// TIA Portal V20 export
FUNCTION "02 T4 LANT HMI" : Void   // FC1212, LAD
TITLE = HMI
{ S7_Optimized_Access := 'TRUE' }
// stored: AutoNumber false, SetENOAutomatically false
BEGIN

REGION Network 1: Reset command interface from HMI in case of time-out
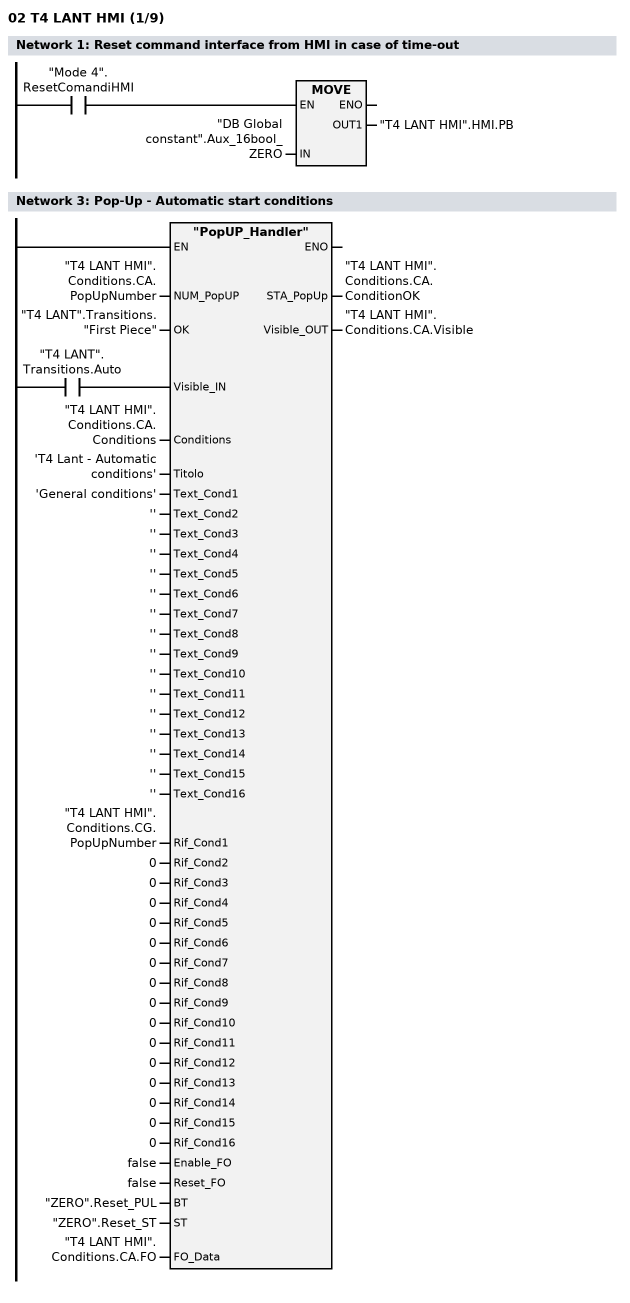
   RUNG wire#powerrail
      Contact( "Mode 4".ResetComandiHMI )
      Move(in := "DB Global constant".Aux_16bool_ZERO, out1 => "T4 LANT HMI".HMI.PB)
   END_RUNG
   // the same network as SCL:
   IF "Mode 4".ResetComandiHMI THEN "T4 LANT HMI".HMI.PB := "DB Global constant".Aux_16bool_ZERO; END_IF;
END_REGION

REGION Network 2: ============ POP UP ============
END_REGION

REGION Network 3: Pop-Up - Automatic start conditions
   RUNG wire#powerrail
      "PopUP_Handler"(Visible_IN := wire#w1, NUM_PopUP := "T4 LANT HMI".Conditions.CA.PopUpNumber, OK := "T4 LANT".Transitions."First Piece", Conditions := "T4 LANT HMI".Conditions.CA.Conditions, Titolo := 'T4 Lant - Automatic conditions', Text_Cond1 := 'General conditions', Text_Cond2 := '', Text_Cond3 := '', Text_Cond4 := '', Text_Cond5 := '', Text_Cond6 := '', Text_Cond7 := '', Text_Cond8 := '', Text_Cond9 := '', Text_Cond10 := '', Text_Cond11 := '', Text_Cond12 := '', Text_Cond13 := '', Text_Cond14 := '', Text_Cond15 := '', Text_Cond16 := '', Rif_Cond1 := "T4 LANT HMI".Conditions.CG.PopUpNumber, Rif_Cond2 := 0, Rif_Cond3 := 0, Rif_Cond4 := 0, Rif_Cond5 := 0, Rif_Cond6 := 0, Rif_Cond7 := 0, Rif_Cond8 := 0, Rif_Cond9 := 0, Rif_Cond10 := 0, Rif_Cond11 := 0, Rif_Cond12 := 0, Rif_Cond13 := 0, Rif_Cond14 := 0, Rif_Cond15 := 0, Rif_Cond16 := 0, Enable_FO := false, Reset_FO := false, BT := "ZERO".Reset_PUL, ST := "ZERO".Reset_ST, FO_Data := "T4 LANT HMI".Conditions.CA.FO, STA_PopUp => "T4 LANT HMI".Conditions.CA.ConditionOK, Visible_OUT => "T4 LANT HMI".Conditions.CA.Visible)
   END_RUNG
   RUNG wire#powerrail
      Contact( "T4 LANT".Transitions.Auto )
   END_RUNG wire#w1
   // the same network as SCL:
   "PopUP_Handler"(NUM_PopUP := "T4 LANT HMI".Conditions.CA.PopUpNumber,
                   OK := "T4 LANT".Transitions."First Piece",
                   Visible_IN := "T4 LANT".Transitions.Auto,
                   Conditions := "T4 LANT HMI".Conditions.CA.Conditions,
                   Titolo := 'T4 Lant - Automatic conditions',
                   Text_Cond1 := 'General conditions',
                   Text_Cond2 := '',
                   Text_Cond3 := '',
                   Text_Cond4 := '',
                   Text_Cond5 := '',
                   Text_Cond6 := '',
                   Text_Cond7 := '',
                   Text_Cond8 := '',
                   Text_Cond9 := '',
                   Text_Cond10 := '',
                   Text_Cond11 := '',
                   Text_Cond12 := '',
                   Text_Cond13 := '',
                   Text_Cond14 := '',
                   Text_Cond15 := '',
                   Text_Cond16 := '',
                   Rif_Cond1 := "T4 LANT HMI".Conditions.CG.PopUpNumber,
                   Rif_Cond2 := 0,
                   Rif_Cond3 := 0,
                   Rif_Cond4 := 0,
                   Rif_Cond5 := 0,
                   Rif_Cond6 := 0,
                   Rif_Cond7 := 0,
                   Rif_Cond8 := 0,
                   Rif_Cond9 := 0,
                   Rif_Cond10 := 0,
                   Rif_Cond11 := 0,
                   Rif_Cond12 := 0,
                   Rif_Cond13 := 0,
                   Rif_Cond14 := 0,
                   Rif_Cond15 := 0,
                   Rif_Cond16 := 0,
                   Enable_FO := false,
                   Reset_FO := false,
                   BT := "ZERO".Reset_PUL,
                   ST := "ZERO".Reset_ST,
                   FO_Data := "T4 LANT HMI".Conditions.CA.FO,
                   STA_PopUp => "T4 LANT HMI".Conditions.CA.ConditionOK,
                   Visible_OUT => "T4 LANT HMI".Conditions.CA.Visible);
END_REGION

REGION Network 4: Pop- Up - General conditions
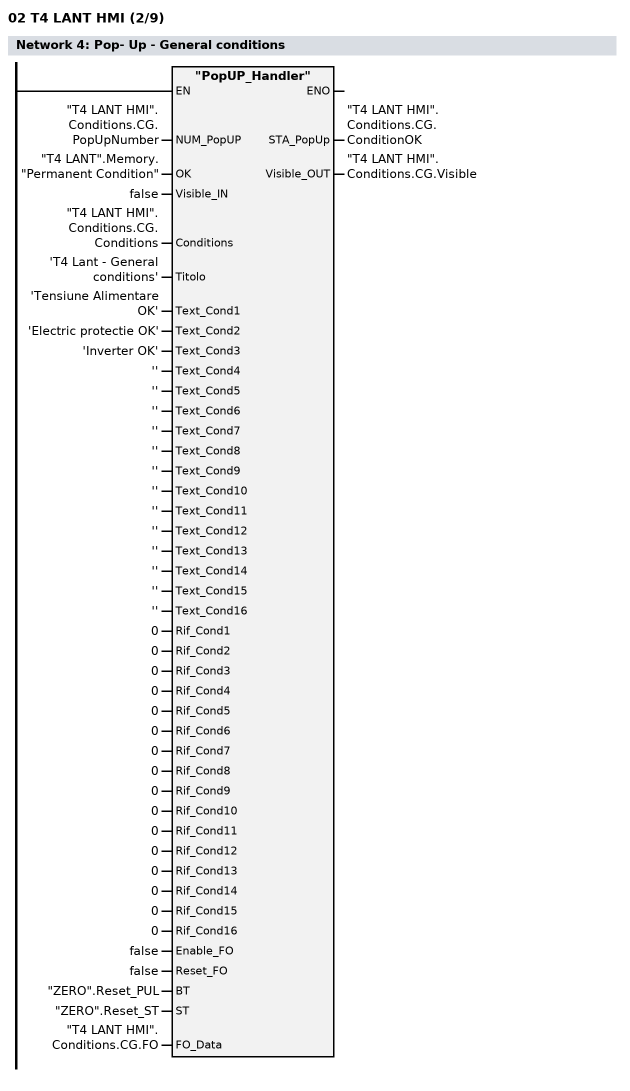
   RUNG wire#powerrail
      "PopUP_Handler"(NUM_PopUP := "T4 LANT HMI".Conditions.CG.PopUpNumber, OK := "T4 LANT".Memory."Permanent Condition", Visible_IN := false, Conditions := "T4 LANT HMI".Conditions.CG.Conditions, Titolo := 'T4 Lant - General conditions', Text_Cond1 := 'Tensiune Alimentare OK', Text_Cond2 := 'Electric protectie OK', Text_Cond3 := 'Inverter OK', Text_Cond4 := '', Text_Cond5 := '', Text_Cond6 := '', Text_Cond7 := '', Text_Cond8 := '', Text_Cond9 := '', Text_Cond10 := '', Text_Cond11 := '', Text_Cond12 := '', Text_Cond13 := '', Text_Cond14 := '', Text_Cond15 := '', Text_Cond16 := '', Rif_Cond1 := 0, Rif_Cond2 := 0, Rif_Cond3 := 0, Rif_Cond4 := 0, Rif_Cond5 := 0, Rif_Cond6 := 0, Rif_Cond7 := 0, Rif_Cond8 := 0, Rif_Cond9 := 0, Rif_Cond10 := 0, Rif_Cond11 := 0, Rif_Cond12 := 0, Rif_Cond13 := 0, Rif_Cond14 := 0, Rif_Cond15 := 0, Rif_Cond16 := 0, Enable_FO := false, Reset_FO := false, BT := "ZERO".Reset_PUL, ST := "ZERO".Reset_ST, FO_Data := "T4 LANT HMI".Conditions.CG.FO, STA_PopUp => "T4 LANT HMI".Conditions.CG.ConditionOK, Visible_OUT => "T4 LANT HMI".Conditions.CG.Visible)
   END_RUNG
   // the same network as SCL:
   "PopUP_Handler"(NUM_PopUP := "T4 LANT HMI".Conditions.CG.PopUpNumber,
                   OK := "T4 LANT".Memory."Permanent Condition",
                   Visible_IN := false,
                   Conditions := "T4 LANT HMI".Conditions.CG.Conditions,
                   Titolo := 'T4 Lant - General conditions',
                   Text_Cond1 := 'Tensiune Alimentare OK',
                   Text_Cond2 := 'Electric protectie OK',
                   Text_Cond3 := 'Inverter OK',
                   Text_Cond4 := '',
                   Text_Cond5 := '',
                   Text_Cond6 := '',
                   Text_Cond7 := '',
                   Text_Cond8 := '',
                   Text_Cond9 := '',
                   Text_Cond10 := '',
                   Text_Cond11 := '',
                   Text_Cond12 := '',
                   Text_Cond13 := '',
                   Text_Cond14 := '',
                   Text_Cond15 := '',
                   Text_Cond16 := '',
                   Rif_Cond1 := 0,
                   Rif_Cond2 := 0,
                   Rif_Cond3 := 0,
                   Rif_Cond4 := 0,
                   Rif_Cond5 := 0,
                   Rif_Cond6 := 0,
                   Rif_Cond7 := 0,
                   Rif_Cond8 := 0,
                   Rif_Cond9 := 0,
                   Rif_Cond10 := 0,
                   Rif_Cond11 := 0,
                   Rif_Cond12 := 0,
                   Rif_Cond13 := 0,
                   Rif_Cond14 := 0,
                   Rif_Cond15 := 0,
                   Rif_Cond16 := 0,
                   Enable_FO := false,
                   Reset_FO := false,
                   BT := "ZERO".Reset_PUL,
                   ST := "ZERO".Reset_ST,
                   FO_Data := "T4 LANT HMI".Conditions.CG.FO,
                   STA_PopUp => "T4 LANT HMI".Conditions.CG.ConditionOK,
                   Visible_OUT => "T4 LANT HMI".Conditions.CG.Visible);
END_REGION

REGION Network 5: PopUP - Cycle start conditions
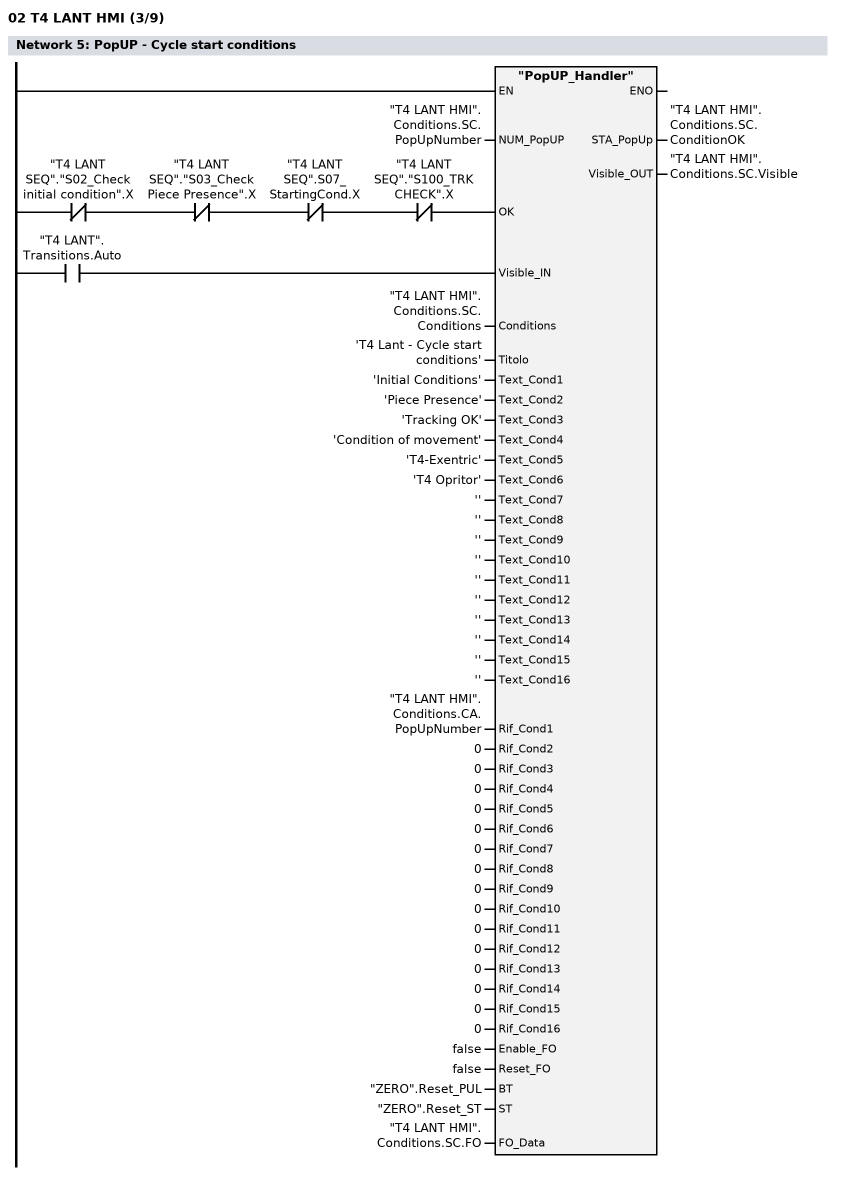
   RUNG wire#powerrail
      "PopUP_Handler"(OK := wire#w1, Visible_IN := wire#w2, NUM_PopUP := "T4 LANT HMI".Conditions.SC.PopUpNumber, Conditions := "T4 LANT HMI".Conditions.SC.Conditions, Titolo := 'T4 Lant - Cycle start conditions', Text_Cond1 := 'Initial Conditions', Text_Cond2 := 'Piece Presence', Text_Cond3 := 'Tracking OK', Text_Cond4 := 'Condition of movement', Text_Cond5 := 'T4-Exentric', Text_Cond6 := 'T4 Opritor', Text_Cond7 := '', Text_Cond8 := '', Text_Cond9 := '', Text_Cond10 := '', Text_Cond11 := '', Text_Cond12 := '', Text_Cond13 := '', Text_Cond14 := '', Text_Cond15 := '', Text_Cond16 := '', Rif_Cond1 := "T4 LANT HMI".Conditions.CA.PopUpNumber, Rif_Cond2 := 0, Rif_Cond3 := 0, Rif_Cond4 := 0, Rif_Cond5 := 0, Rif_Cond6 := 0, Rif_Cond7 := 0, Rif_Cond8 := 0, Rif_Cond9 := 0, Rif_Cond10 := 0, Rif_Cond11 := 0, Rif_Cond12 := 0, Rif_Cond13 := 0, Rif_Cond14 := 0, Rif_Cond15 := 0, Rif_Cond16 := 0, Enable_FO := false, Reset_FO := false, BT := "ZERO".Reset_PUL, ST := "ZERO".Reset_ST, FO_Data := "T4 LANT HMI".Conditions.SC.FO, STA_PopUp => "T4 LANT HMI".Conditions.SC.ConditionOK, Visible_OUT => "T4 LANT HMI".Conditions.SC.Visible)
   END_RUNG
   RUNG wire#powerrail
      I_Contact( "T4 LANT SEQ"."S02_Check initial condition".X )
      I_Contact( "T4 LANT SEQ"."S03_Check Piece Presence".X )
      I_Contact( "T4 LANT SEQ".S07_StartingCond.X )
      I_Contact( "T4 LANT SEQ"."S100_TRK CHECK".X )
   END_RUNG wire#w1
   RUNG wire#powerrail
      Contact( "T4 LANT".Transitions.Auto )
   END_RUNG wire#w2
   // the same network as SCL:
   "PopUP_Handler"(NUM_PopUP := "T4 LANT HMI".Conditions.SC.PopUpNumber,
                   OK := NOT "T4 LANT SEQ"."S02_Check initial condition".X AND NOT "T4 LANT SEQ"."S03_Check Piece Presence".X AND NOT "T4 LANT SEQ".S07_StartingCond.X AND NOT "T4 LANT SEQ"."S100_TRK CHECK".X,
                   Visible_IN := "T4 LANT".Transitions.Auto,
                   Conditions := "T4 LANT HMI".Conditions.SC.Conditions,
                   Titolo := 'T4 Lant - Cycle start conditions',
                   Text_Cond1 := 'Initial Conditions',
                   Text_Cond2 := 'Piece Presence',
                   Text_Cond3 := 'Tracking OK',
                   Text_Cond4 := 'Condition of movement',
                   Text_Cond5 := 'T4-Exentric',
                   Text_Cond6 := 'T4 Opritor',
                   Text_Cond7 := '',
                   Text_Cond8 := '',
                   Text_Cond9 := '',
                   Text_Cond10 := '',
                   Text_Cond11 := '',
                   Text_Cond12 := '',
                   Text_Cond13 := '',
                   Text_Cond14 := '',
                   Text_Cond15 := '',
                   Text_Cond16 := '',
                   Rif_Cond1 := "T4 LANT HMI".Conditions.CA.PopUpNumber,
                   Rif_Cond2 := 0,
                   Rif_Cond3 := 0,
                   Rif_Cond4 := 0,
                   Rif_Cond5 := 0,
                   Rif_Cond6 := 0,
                   Rif_Cond7 := 0,
                   Rif_Cond8 := 0,
                   Rif_Cond9 := 0,
                   Rif_Cond10 := 0,
                   Rif_Cond11 := 0,
                   Rif_Cond12 := 0,
                   Rif_Cond13 := 0,
                   Rif_Cond14 := 0,
                   Rif_Cond15 := 0,
                   Rif_Cond16 := 0,
                   Enable_FO := false,
                   Reset_FO := false,
                   BT := "ZERO".Reset_PUL,
                   ST := "ZERO".Reset_ST,
                   FO_Data := "T4 LANT HMI".Conditions.SC.FO,
                   STA_PopUp => "T4 LANT HMI".Conditions.SC.ConditionOK,
                   Visible_OUT => "T4 LANT HMI".Conditions.SC.Visible);
END_REGION

REGION Network 6: Pop-Up - Conditions of movement FORWARD
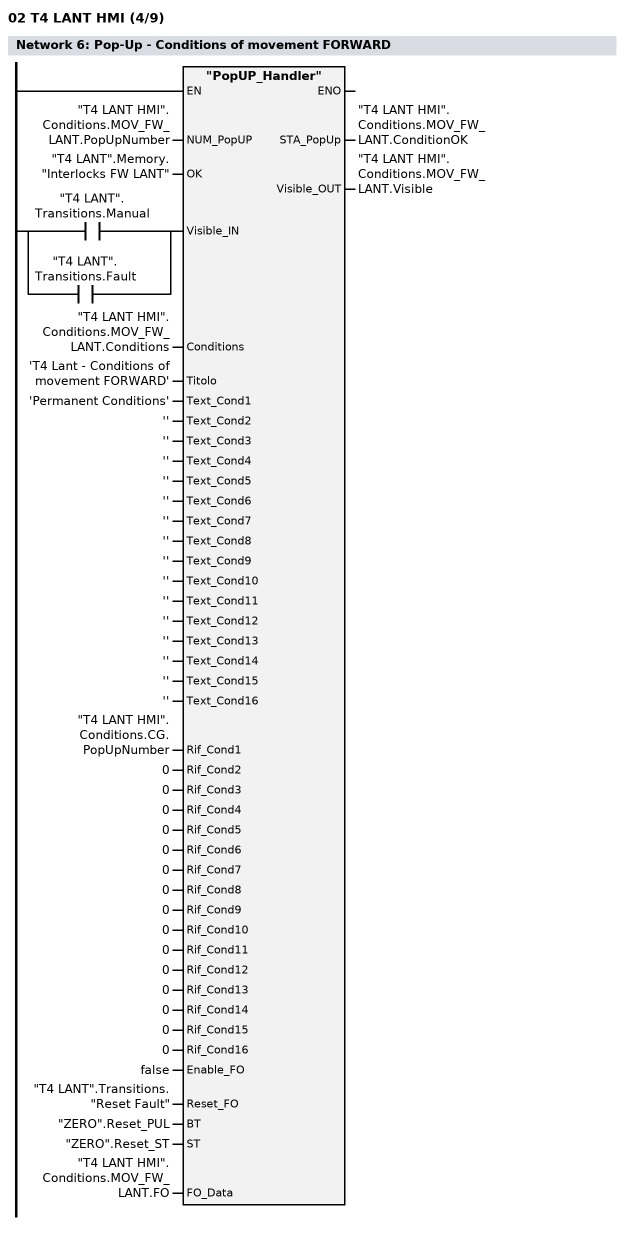
   RUNG wire#powerrail
      "PopUP_Handler"(Visible_IN := wire#w1, NUM_PopUP := "T4 LANT HMI".Conditions.MOV_FW_LANT.PopUpNumber, OK := "T4 LANT".Memory."Interlocks FW LANT", Conditions := "T4 LANT HMI".Conditions.MOV_FW_LANT.Conditions, Titolo := 'T4 Lant - Conditions of movement FORWARD', Text_Cond1 := 'Permanent Conditions', Text_Cond2 := '', Text_Cond3 := '', Text_Cond4 := '', Text_Cond5 := '', Text_Cond6 := '', Text_Cond7 := '', Text_Cond8 := '', Text_Cond9 := '', Text_Cond10 := '', Text_Cond11 := '', Text_Cond12 := '', Text_Cond13 := '', Text_Cond14 := '', Text_Cond15 := '', Text_Cond16 := '', Rif_Cond1 := "T4 LANT HMI".Conditions.CG.PopUpNumber, Rif_Cond2 := 0, Rif_Cond3 := 0, Rif_Cond4 := 0, Rif_Cond5 := 0, Rif_Cond6 := 0, Rif_Cond7 := 0, Rif_Cond8 := 0, Rif_Cond9 := 0, Rif_Cond10 := 0, Rif_Cond11 := 0, Rif_Cond12 := 0, Rif_Cond13 := 0, Rif_Cond14 := 0, Rif_Cond15 := 0, Rif_Cond16 := 0, Enable_FO := false, Reset_FO := "T4 LANT".Transitions."Reset Fault", BT := "ZERO".Reset_PUL, ST := "ZERO".Reset_ST, FO_Data := "T4 LANT HMI".Conditions.MOV_FW_LANT.FO, STA_PopUp => "T4 LANT HMI".Conditions.MOV_FW_LANT.ConditionOK, Visible_OUT => "T4 LANT HMI".Conditions.MOV_FW_LANT.Visible)
   END_RUNG
   RUNG wire#powerrail
      Contact( "T4 LANT".Transitions.Manual )
   END_RUNG wire#w1
   RUNG wire#powerrail
      Contact( "T4 LANT".Transitions.Fault )
   END_RUNG wire#w1
   // the same network as SCL:
   "PopUP_Handler"(NUM_PopUP := "T4 LANT HMI".Conditions.MOV_FW_LANT.PopUpNumber,
                   OK := "T4 LANT".Memory."Interlocks FW LANT",
                   Visible_IN := "T4 LANT".Transitions.Manual OR "T4 LANT".Transitions.Fault,
                   Conditions := "T4 LANT HMI".Conditions.MOV_FW_LANT.Conditions,
                   Titolo := 'T4 Lant - Conditions of movement FORWARD',
                   Text_Cond1 := 'Permanent Conditions',
                   Text_Cond2 := '',
                   Text_Cond3 := '',
                   Text_Cond4 := '',
                   Text_Cond5 := '',
                   Text_Cond6 := '',
                   Text_Cond7 := '',
                   Text_Cond8 := '',
                   Text_Cond9 := '',
                   Text_Cond10 := '',
                   Text_Cond11 := '',
                   Text_Cond12 := '',
                   Text_Cond13 := '',
                   Text_Cond14 := '',
                   Text_Cond15 := '',
                   Text_Cond16 := '',
                   Rif_Cond1 := "T4 LANT HMI".Conditions.CG.PopUpNumber,
                   Rif_Cond2 := 0,
                   Rif_Cond3 := 0,
                   Rif_Cond4 := 0,
                   Rif_Cond5 := 0,
                   Rif_Cond6 := 0,
                   Rif_Cond7 := 0,
                   Rif_Cond8 := 0,
                   Rif_Cond9 := 0,
                   Rif_Cond10 := 0,
                   Rif_Cond11 := 0,
                   Rif_Cond12 := 0,
                   Rif_Cond13 := 0,
                   Rif_Cond14 := 0,
                   Rif_Cond15 := 0,
                   Rif_Cond16 := 0,
                   Enable_FO := false,
                   Reset_FO := "T4 LANT".Transitions."Reset Fault",
                   BT := "ZERO".Reset_PUL,
                   ST := "ZERO".Reset_ST,
                   FO_Data := "T4 LANT HMI".Conditions.MOV_FW_LANT.FO,
                   STA_PopUp => "T4 LANT HMI".Conditions.MOV_FW_LANT.ConditionOK,
                   Visible_OUT => "T4 LANT HMI".Conditions.MOV_FW_LANT.Visible);
END_REGION

REGION Network 7: Pop-Up - Conditions of movement BACKWARD
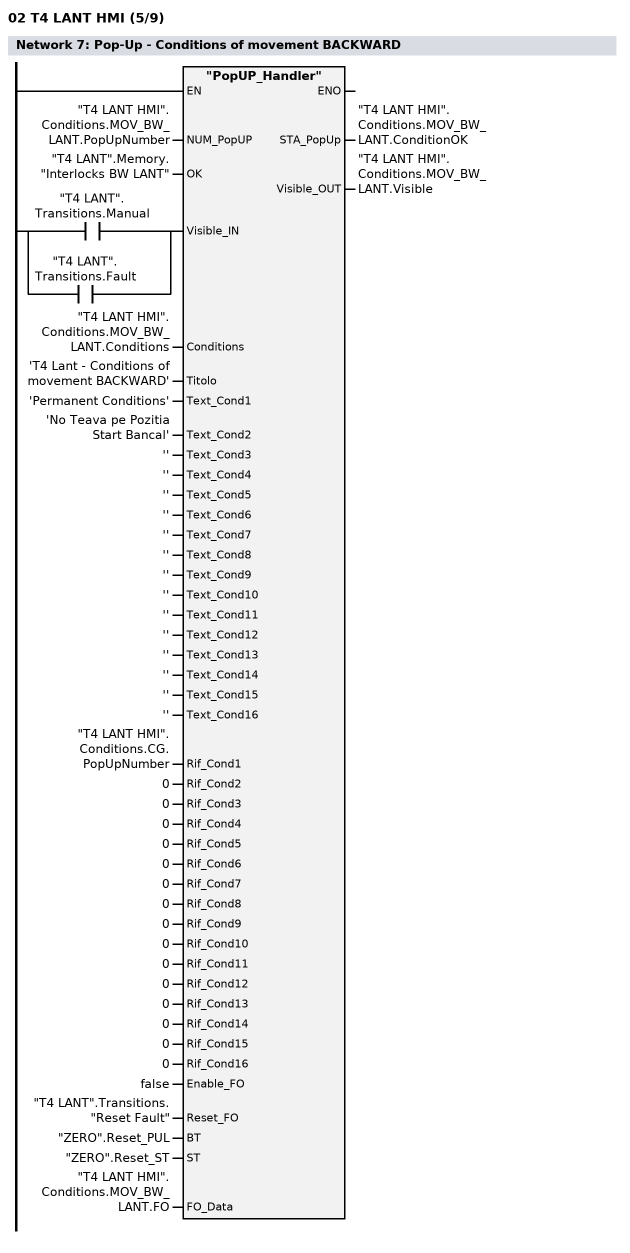
   RUNG wire#powerrail
      "PopUP_Handler"(Visible_IN := wire#w1, NUM_PopUP := "T4 LANT HMI".Conditions.MOV_BW_LANT.PopUpNumber, OK := "T4 LANT".Memory."Interlocks BW LANT", Conditions := "T4 LANT HMI".Conditions.MOV_BW_LANT.Conditions, Titolo := 'T4 Lant - Conditions of movement BACKWARD', Text_Cond1 := 'Permanent Conditions', Text_Cond2 := 'No Teava pe Pozitia Start Bancal', Text_Cond3 := '', Text_Cond4 := '', Text_Cond5 := '', Text_Cond6 := '', Text_Cond7 := '', Text_Cond8 := '', Text_Cond9 := '', Text_Cond10 := '', Text_Cond11 := '', Text_Cond12 := '', Text_Cond13 := '', Text_Cond14 := '', Text_Cond15 := '', Text_Cond16 := '', Rif_Cond1 := "T4 LANT HMI".Conditions.CG.PopUpNumber, Rif_Cond2 := 0, Rif_Cond3 := 0, Rif_Cond4 := 0, Rif_Cond5 := 0, Rif_Cond6 := 0, Rif_Cond7 := 0, Rif_Cond8 := 0, Rif_Cond9 := 0, Rif_Cond10 := 0, Rif_Cond11 := 0, Rif_Cond12 := 0, Rif_Cond13 := 0, Rif_Cond14 := 0, Rif_Cond15 := 0, Rif_Cond16 := 0, Enable_FO := false, Reset_FO := "T4 LANT".Transitions."Reset Fault", BT := "ZERO".Reset_PUL, ST := "ZERO".Reset_ST, FO_Data := "T4 LANT HMI".Conditions.MOV_BW_LANT.FO, STA_PopUp => "T4 LANT HMI".Conditions.MOV_BW_LANT.ConditionOK, Visible_OUT => "T4 LANT HMI".Conditions.MOV_BW_LANT.Visible)
   END_RUNG
   RUNG wire#powerrail
      Contact( "T4 LANT".Transitions.Manual )
   END_RUNG wire#w1
   RUNG wire#powerrail
      Contact( "T4 LANT".Transitions.Fault )
   END_RUNG wire#w1
   // the same network as SCL:
   "PopUP_Handler"(NUM_PopUP := "T4 LANT HMI".Conditions.MOV_BW_LANT.PopUpNumber,
                   OK := "T4 LANT".Memory."Interlocks BW LANT",
                   Visible_IN := "T4 LANT".Transitions.Manual OR "T4 LANT".Transitions.Fault,
                   Conditions := "T4 LANT HMI".Conditions.MOV_BW_LANT.Conditions,
                   Titolo := 'T4 Lant - Conditions of movement BACKWARD',
                   Text_Cond1 := 'Permanent Conditions',
                   Text_Cond2 := 'No Teava pe Pozitia Start Bancal',
                   Text_Cond3 := '',
                   Text_Cond4 := '',
                   Text_Cond5 := '',
                   Text_Cond6 := '',
                   Text_Cond7 := '',
                   Text_Cond8 := '',
                   Text_Cond9 := '',
                   Text_Cond10 := '',
                   Text_Cond11 := '',
                   Text_Cond12 := '',
                   Text_Cond13 := '',
                   Text_Cond14 := '',
                   Text_Cond15 := '',
                   Text_Cond16 := '',
                   Rif_Cond1 := "T4 LANT HMI".Conditions.CG.PopUpNumber,
                   Rif_Cond2 := 0,
                   Rif_Cond3 := 0,
                   Rif_Cond4 := 0,
                   Rif_Cond5 := 0,
                   Rif_Cond6 := 0,
                   Rif_Cond7 := 0,
                   Rif_Cond8 := 0,
                   Rif_Cond9 := 0,
                   Rif_Cond10 := 0,
                   Rif_Cond11 := 0,
                   Rif_Cond12 := 0,
                   Rif_Cond13 := 0,
                   Rif_Cond14 := 0,
                   Rif_Cond15 := 0,
                   Rif_Cond16 := 0,
                   Enable_FO := false,
                   Reset_FO := "T4 LANT".Transitions."Reset Fault",
                   BT := "ZERO".Reset_PUL,
                   ST := "ZERO".Reset_ST,
                   FO_Data := "T4 LANT HMI".Conditions.MOV_BW_LANT.FO,
                   STA_PopUp => "T4 LANT HMI".Conditions.MOV_BW_LANT.ConditionOK,
                   Visible_OUT => "T4 LANT HMI".Conditions.MOV_BW_LANT.Visible);
END_REGION

REGION Network 8: Pop-Up - Conditions of movement Rost FORWARD
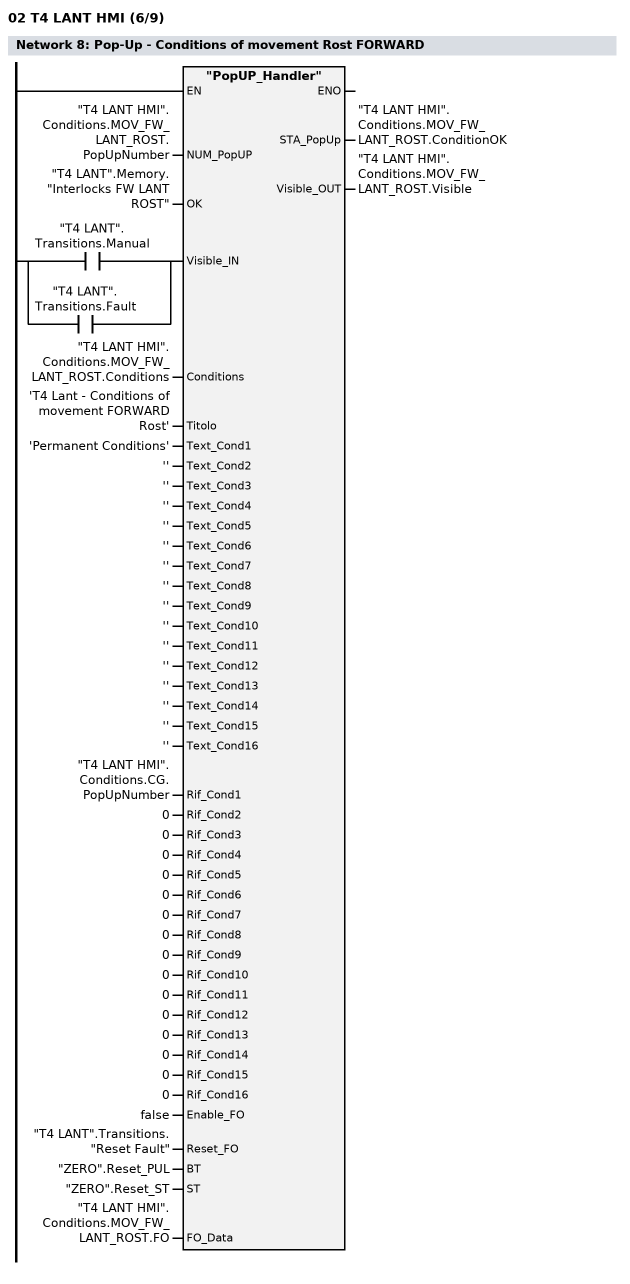
   RUNG wire#powerrail
      "PopUP_Handler"(Visible_IN := wire#w1, NUM_PopUP := "T4 LANT HMI".Conditions.MOV_FW_LANT_ROST.PopUpNumber, OK := "T4 LANT".Memory."Interlocks FW LANT ROST", Conditions := "T4 LANT HMI".Conditions.MOV_FW_LANT_ROST.Conditions, Titolo := 'T4 Lant - Conditions of movement FORWARD Rost', Text_Cond1 := 'Permanent Conditions', Text_Cond2 := '', Text_Cond3 := '', Text_Cond4 := '', Text_Cond5 := '', Text_Cond6 := '', Text_Cond7 := '', Text_Cond8 := '', Text_Cond9 := '', Text_Cond10 := '', Text_Cond11 := '', Text_Cond12 := '', Text_Cond13 := '', Text_Cond14 := '', Text_Cond15 := '', Text_Cond16 := '', Rif_Cond1 := "T4 LANT HMI".Conditions.CG.PopUpNumber, Rif_Cond2 := 0, Rif_Cond3 := 0, Rif_Cond4 := 0, Rif_Cond5 := 0, Rif_Cond6 := 0, Rif_Cond7 := 0, Rif_Cond8 := 0, Rif_Cond9 := 0, Rif_Cond10 := 0, Rif_Cond11 := 0, Rif_Cond12 := 0, Rif_Cond13 := 0, Rif_Cond14 := 0, Rif_Cond15 := 0, Rif_Cond16 := 0, Enable_FO := false, Reset_FO := "T4 LANT".Transitions."Reset Fault", BT := "ZERO".Reset_PUL, ST := "ZERO".Reset_ST, FO_Data := "T4 LANT HMI".Conditions.MOV_FW_LANT_ROST.FO, STA_PopUp => "T4 LANT HMI".Conditions.MOV_FW_LANT_ROST.ConditionOK, Visible_OUT => "T4 LANT HMI".Conditions.MOV_FW_LANT_ROST.Visible)
   END_RUNG
   RUNG wire#powerrail
      Contact( "T4 LANT".Transitions.Manual )
   END_RUNG wire#w1
   RUNG wire#powerrail
      Contact( "T4 LANT".Transitions.Fault )
   END_RUNG wire#w1
   // the same network as SCL:
   "PopUP_Handler"(NUM_PopUP := "T4 LANT HMI".Conditions.MOV_FW_LANT_ROST.PopUpNumber,
                   OK := "T4 LANT".Memory."Interlocks FW LANT ROST",
                   Visible_IN := "T4 LANT".Transitions.Manual OR "T4 LANT".Transitions.Fault,
                   Conditions := "T4 LANT HMI".Conditions.MOV_FW_LANT_ROST.Conditions,
                   Titolo := 'T4 Lant - Conditions of movement FORWARD Rost',
                   Text_Cond1 := 'Permanent Conditions',
                   Text_Cond2 := '',
                   Text_Cond3 := '',
                   Text_Cond4 := '',
                   Text_Cond5 := '',
                   Text_Cond6 := '',
                   Text_Cond7 := '',
                   Text_Cond8 := '',
                   Text_Cond9 := '',
                   Text_Cond10 := '',
                   Text_Cond11 := '',
                   Text_Cond12 := '',
                   Text_Cond13 := '',
                   Text_Cond14 := '',
                   Text_Cond15 := '',
                   Text_Cond16 := '',
                   Rif_Cond1 := "T4 LANT HMI".Conditions.CG.PopUpNumber,
                   Rif_Cond2 := 0,
                   Rif_Cond3 := 0,
                   Rif_Cond4 := 0,
                   Rif_Cond5 := 0,
                   Rif_Cond6 := 0,
                   Rif_Cond7 := 0,
                   Rif_Cond8 := 0,
                   Rif_Cond9 := 0,
                   Rif_Cond10 := 0,
                   Rif_Cond11 := 0,
                   Rif_Cond12 := 0,
                   Rif_Cond13 := 0,
                   Rif_Cond14 := 0,
                   Rif_Cond15 := 0,
                   Rif_Cond16 := 0,
                   Enable_FO := false,
                   Reset_FO := "T4 LANT".Transitions."Reset Fault",
                   BT := "ZERO".Reset_PUL,
                   ST := "ZERO".Reset_ST,
                   FO_Data := "T4 LANT HMI".Conditions.MOV_FW_LANT_ROST.FO,
                   STA_PopUp => "T4 LANT HMI".Conditions.MOV_FW_LANT_ROST.ConditionOK,
                   Visible_OUT => "T4 LANT HMI".Conditions.MOV_FW_LANT_ROST.Visible);
END_REGION

REGION Network 9: Pop-Up - Conditions of movement Rost BACKWARD
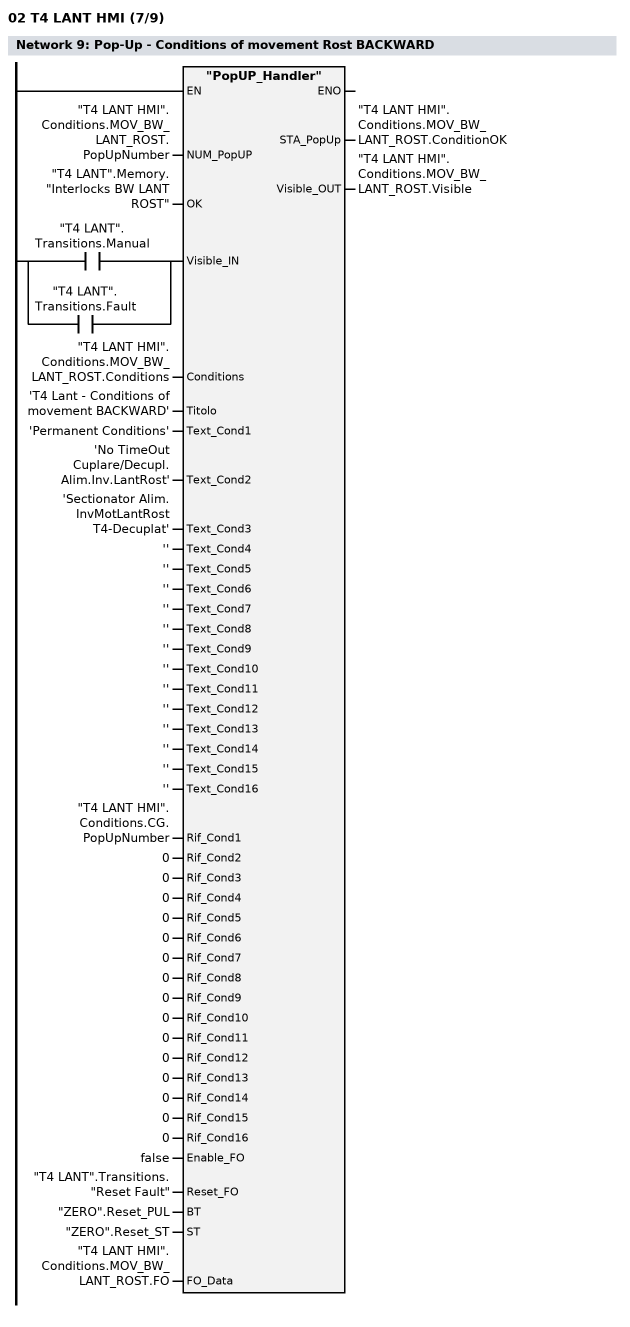
   RUNG wire#powerrail
      "PopUP_Handler"(Visible_IN := wire#w1, NUM_PopUP := "T4 LANT HMI".Conditions.MOV_BW_LANT_ROST.PopUpNumber, OK := "T4 LANT".Memory."Interlocks BW LANT ROST", Conditions := "T4 LANT HMI".Conditions.MOV_BW_LANT_ROST.Conditions, Titolo := 'T4 Lant - Conditions of movement BACKWARD', Text_Cond1 := 'Permanent Conditions', Text_Cond2 := 'No TimeOut Cuplare/Decupl. Alim.Inv.LantRost', Text_Cond3 := 'Sectionator Alim. InvMotLantRost T4-Decuplat', Text_Cond4 := '', Text_Cond5 := '', Text_Cond6 := '', Text_Cond7 := '', Text_Cond8 := '', Text_Cond9 := '', Text_Cond10 := '', Text_Cond11 := '', Text_Cond12 := '', Text_Cond13 := '', Text_Cond14 := '', Text_Cond15 := '', Text_Cond16 := '', Rif_Cond1 := "T4 LANT HMI".Conditions.CG.PopUpNumber, Rif_Cond2 := 0, Rif_Cond3 := 0, Rif_Cond4 := 0, Rif_Cond5 := 0, Rif_Cond6 := 0, Rif_Cond7 := 0, Rif_Cond8 := 0, Rif_Cond9 := 0, Rif_Cond10 := 0, Rif_Cond11 := 0, Rif_Cond12 := 0, Rif_Cond13 := 0, Rif_Cond14 := 0, Rif_Cond15 := 0, Rif_Cond16 := 0, Enable_FO := false, Reset_FO := "T4 LANT".Transitions."Reset Fault", BT := "ZERO".Reset_PUL, ST := "ZERO".Reset_ST, FO_Data := "T4 LANT HMI".Conditions.MOV_BW_LANT_ROST.FO, STA_PopUp => "T4 LANT HMI".Conditions.MOV_BW_LANT_ROST.ConditionOK, Visible_OUT => "T4 LANT HMI".Conditions.MOV_BW_LANT_ROST.Visible)
   END_RUNG
   RUNG wire#powerrail
      Contact( "T4 LANT".Transitions.Manual )
   END_RUNG wire#w1
   RUNG wire#powerrail
      Contact( "T4 LANT".Transitions.Fault )
   END_RUNG wire#w1
   // the same network as SCL:
   "PopUP_Handler"(NUM_PopUP := "T4 LANT HMI".Conditions.MOV_BW_LANT_ROST.PopUpNumber,
                   OK := "T4 LANT".Memory."Interlocks BW LANT ROST",
                   Visible_IN := "T4 LANT".Transitions.Manual OR "T4 LANT".Transitions.Fault,
                   Conditions := "T4 LANT HMI".Conditions.MOV_BW_LANT_ROST.Conditions,
                   Titolo := 'T4 Lant - Conditions of movement BACKWARD',
                   Text_Cond1 := 'Permanent Conditions',
                   Text_Cond2 := 'No TimeOut Cuplare/Decupl. Alim.Inv.LantRost',
                   Text_Cond3 := 'Sectionator Alim. InvMotLantRost T4-Decuplat',
                   Text_Cond4 := '',
                   Text_Cond5 := '',
                   Text_Cond6 := '',
                   Text_Cond7 := '',
                   Text_Cond8 := '',
                   Text_Cond9 := '',
                   Text_Cond10 := '',
                   Text_Cond11 := '',
                   Text_Cond12 := '',
                   Text_Cond13 := '',
                   Text_Cond14 := '',
                   Text_Cond15 := '',
                   Text_Cond16 := '',
                   Rif_Cond1 := "T4 LANT HMI".Conditions.CG.PopUpNumber,
                   Rif_Cond2 := 0,
                   Rif_Cond3 := 0,
                   Rif_Cond4 := 0,
                   Rif_Cond5 := 0,
                   Rif_Cond6 := 0,
                   Rif_Cond7 := 0,
                   Rif_Cond8 := 0,
                   Rif_Cond9 := 0,
                   Rif_Cond10 := 0,
                   Rif_Cond11 := 0,
                   Rif_Cond12 := 0,
                   Rif_Cond13 := 0,
                   Rif_Cond14 := 0,
                   Rif_Cond15 := 0,
                   Rif_Cond16 := 0,
                   Enable_FO := false,
                   Reset_FO := "T4 LANT".Transitions."Reset Fault",
                   BT := "ZERO".Reset_PUL,
                   ST := "ZERO".Reset_ST,
                   FO_Data := "T4 LANT HMI".Conditions.MOV_BW_LANT_ROST.FO,
                   STA_PopUp => "T4 LANT HMI".Conditions.MOV_BW_LANT_ROST.ConditionOK,
                   Visible_OUT => "T4 LANT HMI".Conditions.MOV_BW_LANT_ROST.Visible);
END_REGION

REGION Network 10: ============ HMI STATE ============
END_REGION

REGION Network 11: HMI Status - Mod Operare
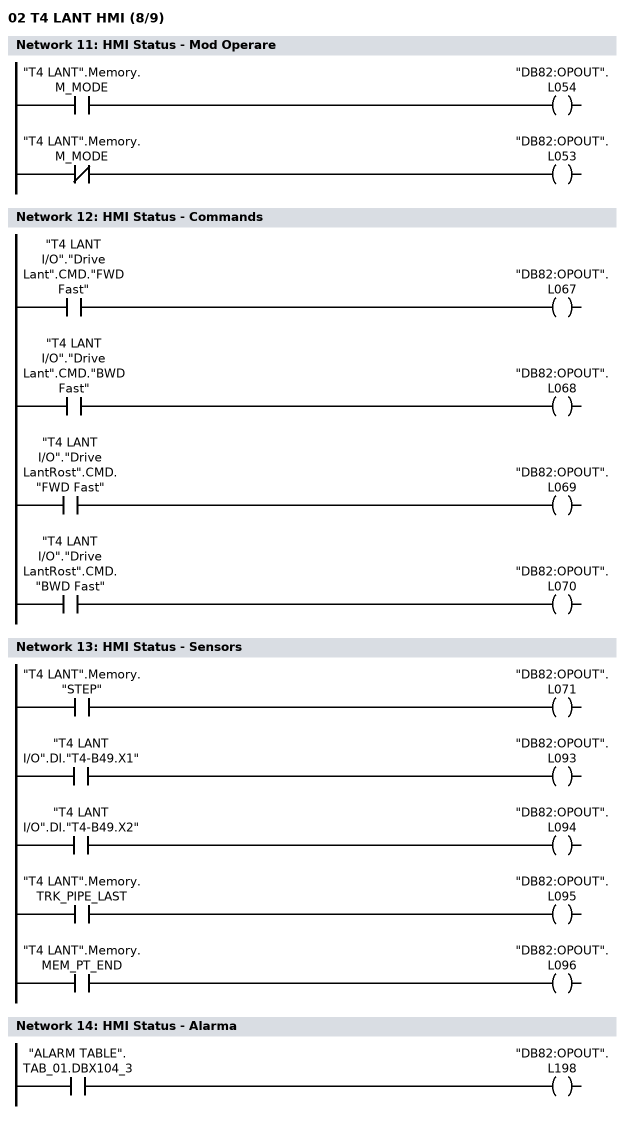
   RUNG wire#powerrail
      Contact( "T4 LANT".Memory.M_MODE )
      Coil( "DB82:OPOUT".L054 )
   END_RUNG
   RUNG wire#powerrail
      I_Contact( "T4 LANT".Memory.M_MODE )
      Coil( "DB82:OPOUT".L053 )
   END_RUNG
   // the same network as SCL:
   "DB82:OPOUT".L054 := "T4 LANT".Memory.M_MODE;
   "DB82:OPOUT".L053 := NOT "T4 LANT".Memory.M_MODE;
END_REGION

REGION Network 12: HMI Status - Commands
   RUNG wire#powerrail
      Contact( "T4 LANT I/O"."Drive Lant".CMD."FWD Fast" )
      Coil( "DB82:OPOUT".L067 )
   END_RUNG
   RUNG wire#powerrail
      Contact( "T4 LANT I/O"."Drive Lant".CMD."BWD Fast" )
      Coil( "DB82:OPOUT".L068 )
   END_RUNG
   RUNG wire#powerrail
      Contact( "T4 LANT I/O"."Drive LantRost".CMD."FWD Fast" )
      Coil( "DB82:OPOUT".L069 )
   END_RUNG
   RUNG wire#powerrail
      Contact( "T4 LANT I/O"."Drive LantRost".CMD."BWD Fast" )
      Coil( "DB82:OPOUT".L070 )
   END_RUNG
   // the same network as SCL:
   "DB82:OPOUT".L067 := "T4 LANT I/O"."Drive Lant".CMD."FWD Fast";
   "DB82:OPOUT".L068 := "T4 LANT I/O"."Drive Lant".CMD."BWD Fast";
   "DB82:OPOUT".L069 := "T4 LANT I/O"."Drive LantRost".CMD."FWD Fast";
   "DB82:OPOUT".L070 := "T4 LANT I/O"."Drive LantRost".CMD."BWD Fast";
END_REGION

REGION Network 13: HMI Status - Sensors
   RUNG wire#powerrail
      Contact( "T4 LANT".Memory."STEP" )
      Coil( "DB82:OPOUT".L071 )
   END_RUNG
   RUNG wire#powerrail
      Contact( "T4 LANT I/O".DI."T4-B49.X1" )
      Coil( "DB82:OPOUT".L093 )
   END_RUNG
   RUNG wire#powerrail
      Contact( "T4 LANT I/O".DI."T4-B49.X2" )
      Coil( "DB82:OPOUT".L094 )
   END_RUNG
   RUNG wire#powerrail
      Contact( "T4 LANT".Memory.TRK_PIPE_LAST )
      Coil( "DB82:OPOUT".L095 )
   END_RUNG
   RUNG wire#powerrail
      Contact( "T4 LANT".Memory.MEM_PT_END )
      Coil( "DB82:OPOUT".L096 )
   END_RUNG
   // the same network as SCL:
   "DB82:OPOUT".L071 := "T4 LANT".Memory."STEP";
   "DB82:OPOUT".L093 := "T4 LANT I/O".DI."T4-B49.X1";
   "DB82:OPOUT".L094 := "T4 LANT I/O".DI."T4-B49.X2";
   "DB82:OPOUT".L095 := "T4 LANT".Memory.TRK_PIPE_LAST;
   "DB82:OPOUT".L096 := "T4 LANT".Memory.MEM_PT_END;
END_REGION

REGION Network 14: HMI Status - Alarma
   RUNG wire#powerrail
      Contact( "ALARM TABLE".TAB_01.DBX104_3 )
      Coil( "DB82:OPOUT".L198 )
   END_RUNG
   // the same network as SCL:
   "DB82:OPOUT".L198 := "ALARM TABLE".TAB_01.DBX104_3;
END_REGION

REGION Network 15: Device status
   // m0.7 comandi uscite
   // M0.7 minimun energy conditions
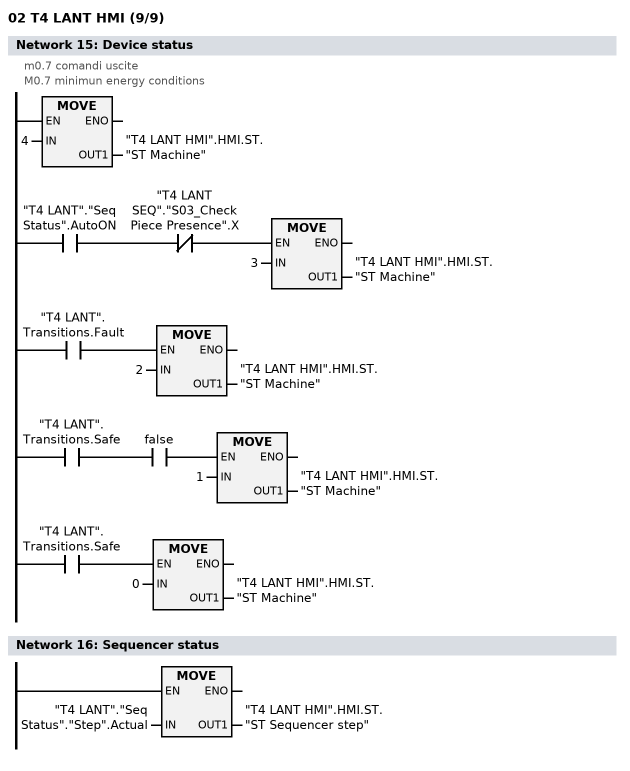
   RUNG wire#powerrail
      Move(in := 4, out1 => "T4 LANT HMI".HMI.ST."ST Machine")
   END_RUNG
   RUNG wire#powerrail
      Contact( "T4 LANT"."Seq Status".AutoON )
      I_Contact( "T4 LANT SEQ"."S03_Check Piece Presence".X )
      Move(in := 3, out1 => "T4 LANT HMI".HMI.ST."ST Machine")
   END_RUNG
   RUNG wire#powerrail
      Contact( "T4 LANT".Transitions.Fault )
      Move(in := 2, out1 => "T4 LANT HMI".HMI.ST."ST Machine")
   END_RUNG
   RUNG wire#powerrail
      Contact( "T4 LANT".Transitions.Safe )
      Contact( false )
      Move(in := 1, out1 => "T4 LANT HMI".HMI.ST."ST Machine")
   END_RUNG
   RUNG wire#powerrail
      Contact( "T4 LANT".Transitions.Safe )
      Move(in := 0, out1 => "T4 LANT HMI".HMI.ST."ST Machine")
   END_RUNG
   // the same network as SCL:
   "T4 LANT HMI".HMI.ST."ST Machine" := 4;
   IF "T4 LANT"."Seq Status".AutoON AND NOT "T4 LANT SEQ"."S03_Check Piece Presence".X THEN
       "T4 LANT HMI".HMI.ST."ST Machine" := 3;
   END_IF;
   IF "T4 LANT".Transitions.Fault THEN "T4 LANT HMI".HMI.ST."ST Machine" := 2; END_IF;
   IF "T4 LANT".Transitions.Safe AND false THEN "T4 LANT HMI".HMI.ST."ST Machine" := 1; END_IF;
   IF "T4 LANT".Transitions.Safe THEN "T4 LANT HMI".HMI.ST."ST Machine" := 0; END_IF;
END_REGION

REGION Network 16: Sequencer status
   RUNG wire#powerrail
      Move(in := "T4 LANT"."Seq Status"."Step".Actual, out1 => "T4 LANT HMI".HMI.ST."ST Sequencer step")
   END_RUNG
   // the same network as SCL:
   "T4 LANT HMI".HMI.ST."ST Sequencer step" := "T4 LANT"."Seq Status"."Step".Actual;
END_REGION
END_FUNCTION
